FUNCTION_BLOCK FB_UpperFeedInConveyor EXTENDS FB_ObjectBase_V2
VAR_INPUT
	
	_fbDiameterMovement : REFERENCE TO FB_DiameterMovement;
	
	Cylinder 	: REFERENCE TO UNI_CylinderList;
	Motor	 	: REFERENCE TO UNI_MotorList;
	Input 	 	: REFERENCE TO ST_InputTable;
	OutPut	 	: REFERENCE TO ST_OutputTable;
	
	Info		: ST_Auto_UpperFeedInConveyorInfo;
	
	AddingBox	: BOOL;
//    Execute    :BOOL;   // True : This prog will start.
//    Abort      :BOOL;   // True : This prog will be abort.
//    Reset      :BOOL;   // True : This prog will be reset.
//    ObjectName :STRING; // Set this fb name(About it's action)
END_VAR

VAR_OUTPUT
//	Status		: ST_StatusBasic;
	FeedBack    : ST_Auto_UpperFeedInConveyorFeedback;	
	_bForceUpperCV_Use	: BOOL;	
//    Busy    :BOOL;        // True : This prog is running.
//    Done    :BOOL;        // True : Command has been executed.
//    Aborted :BOOL;        // True : This prog is aborted.
//    Error   :BOOL;        // True : This prog has an error.
//    ErrorID :UINT;       // Output ErrorID
//    Status  :T_MaxString; // Output this prog status by string(255bytes)
END_VAR

VAR
//    eState :E_MethodStatus_Basic;
//	uiExecutingStep : UDINT; // This var is used to been controll STATE_EXECUTING process.
//	uiResettingStep : UDINT;
//	uiAbortingStep : UDINT;
//	_Executed :BOOL; // Executing process completed.
//	_Error : BOOL; // FB has an error.
//	_ResetCompleted : BOOL; // FB resetting completed.
//	_AbortCompleted : BOOL; // FB aborting completed.
	_Abort		: BOOL;
	strStatus	: T_MaxString;
	uiResumeStep : UINT;
	iMoveConveyor	:INT;// 1 = MoveForward , -1 = Move reverse , 0 or other = Stop
	tonUpperConveyorTimeOut			:TON;
	tonUpperConveyorDelay			:TON;
	tonUpperTimeOut					:TON;
	tonUpperTimeOutFive 			:TON;
	tonWaitSecondBoxArriveTimeout 	:TON;
	tonFeedAirBlowtime 				:TON;
	tonReverseConveyorDelay			:TON;
	TON_CheckHaveBox				:TON ;
	NoFirstBoxDiameter : BOOL;
	SecondBox	:BOOL;
	bSecondBoxInCameraPos :BOOL;
	uiFirstBoxDiameterStep :UINT :=0;
	uiSecondBoxAirBlowStep :UINT :=0;
	_UniqueErrorCode :STRING;
	
	
	//record time for C# photo
	tRecordTimer 		: ARRAY [1..100] OF TIME;
	tRecordFirstTimer	: ARRAY [1..100] OF TIME;
	tRecordSecondTimer	: ARRAY [1..100] OF TIME;
	TON_RecordTimer 	: TON;
	TON_RecordFirstTimer		: TON ;
	TON_RecordSecondTimer		: TON;
	TSaveTime					: TIME;
	TSaveFirstTime				: TIME;
	TSaveSecondTime				: TIME;
	iArrayNumber 				: INT :=1;
	iResetNumber				: INT;
	bResetRecordInfo			: BOOL;
	
	
END_VAR

A00_BasicUnits();
SUPER^.A10_StateControl();

ACTION A00_BasicUnits:
tonUpperConveyorTimeOut(PT:=T#20S);
tonUpperConveyorDelay();
tonUpperTimeOut(PT:=T#5.0S);
tonUpperTimeOutfive(PT:=T#60S);
tonWaitSecondBoxArriveTimeout(PT:=T#20S);
tonFeedAirBlowtime(PT:=info.FeedAirblowTime);
tonReverseConveyorDelay(PT:=T#6S);
TON_CheckHaveBox(PT :=T#35S);
ErrorID :=2710;



TON_RecordTimer (PT:=T#1D);
TON_RecordFirstTimer (PT := T#1D);
TON_RecordSecondTimer (PT := T#1D);

// only for record the photo time use
IF bResetRecordInfo THEN
	FOR iResetNumber :=1 TO 100 DO
		tRecordTimer[iResetNumber] :=T#0S;
		tRecordFirstTimer[iResetNumber] :=T#0S;
		tRecordSecondTimer[iResetNumber] :=T#0S;
	END_FOR
END_IF
END_ACTION

METHOD GetModelState
VAR_OUTPUT
    xDone    :BOOL;
    xBusy    :BOOL;
    xError   :BOOL;
    xAborted :BOOL;
    iErrorID :UDINT;
	UniqueErrorCode : STRING;
END_VAR
xDone    := Done;
xBusy    := Busy;
xError   := Error;
xAborted := Abort;
iErrorID := ErrorID;
END_METHOD

METHOD GetName : STRING
GetName := ObjectName;
END_METHOD

METHOD  M_STATE_ABORTED
VAR_INPUT
END_VAR
ERROR :=TRUE;
Busy := FALSE;
Aborted := TRUE;
_Abort := FALSE;
UniqueErrorCode:=_UniqueErrorCode;
SUPER^.Status := strStatus;

IF NOT Execute THEN
	eSTATE:=STATE_RESETTING;
	
ELSIF Execute AND Reset THEN

		CASE uiExecutingStep OF
			20:
				uiExecutingStep :=10;
				strStatus :='prepare cylinders retry';
				
			100:
				uiExecutingStep :=100;
				strStatus :='check no box retry';
			200:
				uiExecutingStep :=200;
				strStatus :='check Block3Cylinder retry';

			400://將讀碼壓盒1 往後 重做一次
				Cylinder.List.fbUpCV_CamaraPress1.M_Retract();
				IF Cylinder.List.fbUpCV_CamaraPress1.InRearPosition THEN
				uiExecutingStep :=300;
				strStatus :='check ReadCodeBox1 infrontposition retry';
				END_IF
			460:	//Box1 done step abort
				uiExecutingStep :=450;
				strStatus :='Check FirstBoxCamaraDone info retry';
			550:
				uiExecutingStep :=500;
				strStatus :='ReadCodePressBox1Cylinder and FeedInBlockBox3Cylinder Backward retry';
			600:
				uiExecutingStep :=600;
				strStatus :='FirstBoxCameraDiameterRequest Info retry';
			610:
				uiExecutingStep :=610;
				strStatus :='CodeReadingBoxDetection first box leave retry';
			700:
				uiExecutingStep :=700;
				strStatus :='UpperFeedInBlockBox2Cylinder MoveForward retry';
			800:
				uiExecutingStep :=800;
				strStatus :='Box not at UpperBox2Detection retry ';
				
			1000:
				Cylinder.List.fbUpCV_DiameterPress.M_Retract();
				IF Cylinder.List.fbUpCV_DiameterPress.InRearPosition THEN
					uiExecutingStep :=800;
					strStatus :='DiameterMeasurementPressBoxCylinder MoveBackward retry';
				END_IF
			1200:
				Cylinder.List.fbUpCV_CamaraPress1.M_Retract();
				Cylinder.List.fbUpCV_CamaraPress2.M_Retract();
				IF Cylinder.List.fbUpCV_CamaraPress1.InRearPosition AND 
					Cylinder.List.fbUpCV_CamaraPress2.InRearPosition THEN
					uiExecutingStep :=1100;
					strStatus :='ReadCodePressBox 1 and 2 Cylinder retry';
				END_IF
			1300:
				uiExecutingStep :=1300;
				strStatus :='SecondBoxCameraDone info retry';
			1400:
				uiExecutingStep :=1400;
				strStatus :='FirstBoxCameraDiameterDone info retry';
			1600:
				uiExecutingStep :=1500;
				strStatus :='DiameterMeasurementPressBoxCylinder and FeedInBlockBox2Cylinder MoveBackward retry';
			1700:
				uiExecutingStep :=1700;
				strStatus :='check UpperBox2Detection have box';
			1800:
				Cylinder.List.fbUpCV_DiameterPress.M_Retract();
				IF Cylinder.List.fbUpCV_DiameterPress.InRearPosition THEN
				uiExecutingStep :=1700;
				strStatus :='DiameterMeasurementPressBoxCylinder Forward retry';
				END_IF
			1900:
				uiExecutingStep :=1900;
				strStatus :='DiameterMovement PickDone  retry';
			2000:
				uiExecutingStep :=2000;
				strStatus :='SecondBoxCameraDiameterDone retry';
			2100:	
				uiExecutingStep :=2100;
				strStatus :='_fbDiameterMovement done retry';
			2200:
				
				
		END_CASE
	
	eSTATE:=STATE_EXECUTING;
	
END_IF
END_METHOD

METHOD  M_STATE_ABORTING
VAR_INPUT
END_VAR
Busy :=FALSE;
CASE uiAbortingStep OF
	0:
		tonUpperConveyorTimeOut.IN 	:=FALSE;
		tonUpperConveyorDelay.IN	:=FALSE;
		tonUpperTimeOut.IN 			:=FALSE;
		tonUpperTimeOutfive.IN		:=FALSE;
		TON_CheckHaveBox.IN 		:=FALSE;
		uiAbortingStep :=100;
	100:
		Motor.List.UpCV.M_MotorStop();
		OutPut.bCamara_Blow :=FALSE;
		IF Motor.List.UpCV.InStopped THEN
			uiAbortingStep :=9999;
		END_IF
	9999:	
		_AbortCompleted:=TRUE;
END_CASE

IF _AbortCompleted THEN	
	eSTATE :=STATE_ABORTED;
END_IF
END_METHOD

METHOD  M_STATE_DONE
VAR_INPUT
END_VAR
Busy := FALSE;
Done:=TRUE;
_fbDiameterMovement.Execute := FALSE;
_fbDiameterMovement.bContinue:=FALSE;
IF NOT Execute THEN
	eSTATE:=STATE_RESETTING;
END_IF
END_METHOD

METHOD  M_STATE_DORMANT
VAR_INPUT
END_VAR
Busy    := FALSE;
Done    := FALSE;
Aborted := FALSE;
Error   := FALSE;
FeedBack.InterventionRequest :=FALSE;
strStatus :='No Error';
uiExecutingStep :=0;
uiResettingStep	:=0;
NoFirstBoxDiameter:= SecondBox:=FALSE;
tonUpperConveyorTimeOut.IN := FALSE;
tonUpperConveyorDelay.IN :=FALSE;
tonUpperTimeOut.IN :=FALSE;
tonUpperTimeOutFive.IN :=FALSE;
tonWaitSecondBoxArriveTimeout.IN :=FALSE;
TON_CheckHaveBox.IN :=false;
tonFeedAirBlowtime.IN :=false;
bSecondBoxInCameraPos := FALSE;
_bForceUpperCV_Use := false;
_Abort := _Executed := _Error:= _ResetCompleted:=_AbortCompleted:=FALSE;
iMoveConveyor := 0;
uiFirstBoxDiameterStep  :=0;
uiSecondBoxAirBlowStep	:=0;
_UniqueErrorCode :='0';
IF Execute THEN
	eSTATE:=STATE_EXECUTING;
END_IF
END_METHOD

METHOD  M_STATE_ERROR
VAR_INPUT
END_VAR
ERROR :=TRUE;
Busy :=FALSE;
UniqueErrorCode:=_UniqueErrorCode;
SUPER^.Status := strStatus;
_fbDiameterMovement.Execute := FALSE;


Motor.List.UpCV.M_MotorStop(); 
OutPut.bCamara_Blow :=FALSE;

IF NOT Execute THEN	
eSTATE:=STATE_RESETTING;
END_IF
END_METHOD

METHOD  M_STATE_EXECUTING
VAR_INPUT
END_VAR

VAR_INST
	
	
END_VAR
VAR
	END_I: INT;
	
END_VAR
Busy :=TRUE;

//Conveyor motor control
CASE iMoveConveyor OF
	1:
	Motor.list.UpCV.M_MoveForward();
	Cylinder.List.fbUpCV_CamaraPress4.M_Retract(); //Feedin working , open the end to allow box feedin
	//OutPut.bCamara_Blow :=TRUE;
	-1:
	Motor.list.UpCV.M_MoveBackward();
	Cylinder.List.fbUpCV_CamaraPress4.M_Retract(); //Feedin working , open the end to allow box feedin
ELSE		
	Motor.list.UpCV.M_MotorStop();
	Cylinder.List.fbUpCV_CamaraPress4.M_Extend();// End feedin , block the conveyor in case no one push boxes in working area
	//OutPut.bCamara_Blow :=FALSE;		change use airflow to take photo before
END_CASE



CASE uiExecutingStep OF
	
0 : // StandBy
	TON_RecordTimer.IN := TRUE;
	iMoveConveyor:=0;
	tonUpperConveyorTimeOut.IN:=FALSE;
	tonUpperConveyorDelay.IN :=FALSE;
	tonUpperConveyorDelay.PT:=T#200MS;
	IF Info.NrOfBox=1 THEN
		SecondBox:=FALSE;
	ELSIF Info.NrOfBox=2 THEN
		SecondBox:=TRUE;	
	ELSE
	_Error := TRUE;
	  strStatus := 'Data not correct';		
	END_IF
	uiExecutingStep :=10;

10: //Prepare cylinders
	IF Cylinder.List.fbUpCV_FeedInPress1.xError THEN
		Cylinder.List.fbUpCV_FeedInPress1.M_Reset();
	END_IF
	IF Cylinder.List.fbUpCV_FeedInPress2.xError THEN
		Cylinder.List.fbUpCV_FeedInPress1.M_Reset();
	END_IF
	IF Cylinder.List.fbUpCV_DiameterPress.xError THEN
		Cylinder.List.fbUpCV_DiameterPress.M_Reset();
	END_IF
	IF Cylinder.List.fbUpCV_CamaraPress1.xError THEN
		Cylinder.List.fbUpCV_CamaraPress1.M_Reset();
	END_IF
	IF Cylinder.List.fbUpCV_CamaraPress2.xError THEN
		Cylinder.List.fbUpCV_CamaraPress2.M_Reset();
	END_IF
	IF Cylinder.List.fbUpCV_CamaraPress4.xError THEN
		Cylinder.List.fbUpCV_CamaraPress4.M_Reset();
	END_IF
	IF Cylinder.List.fbUpCV_Block1.xError THEN
		Cylinder.List.fbUpCV_Block1.M_Reset();
	END_IF
	IF Cylinder.List.fbUpCV_Block2.xError THEN
		Cylinder.List.fbUpCV_Block2.M_Reset();
	END_IF
	IF Cylinder.List.fbUpCV_Block3.xError THEN
		Cylinder.List.fbUpCV_Block3.M_Reset();
	END_IF
	IF Motor.List.UpCV.xError THEN
		Motor.List.UpCV.M_Reset();
	END_IF
	
	uiExecutingStep :=20;
	
20: //Prepare cylinders
	tonUpperTimeOut.IN :=TRUE;
	Cylinder.List.fbUpCV_FeedInPress1.M_Retract();		(* Cylinder.List.fbUpCV_FeedInPress1.M_Retract();*)	
	Cylinder.List.fbUpCV_FeedInPress2.M_Retract();		(*Cylinder.List.fbUpCV_FeedInPress2.M_Retract();*)
	Cylinder.List.fbUpCV_DiameterPress.M_Retract();		(*Cylinder.List.fbUpCV_DiameterPress.M_Retract();*)
	Cylinder.List.fbUpCV_CamaraPress1.M_Retract();		(*Cylinder.List.fbUpCV_CamaraPress1.M_Retract();*)		
	//Cylinder.List.fbUpCV_CamaraPress2.M_Retract();	(*Cylinder.List.fbUpCV_CamaraPress2.M_Retract();*)
	Cylinder.List.fbUpCV_CamaraPress4.M_Retract();		(*Cylinder.List.fbUpCV_CamaraPress4.M_Retract();*)	
	Cylinder.List.fbUpCV_Block1.M_Retract();			(*Cylinder.List.fbUpCV_Block1.M_Retract();*)
	Cylinder.List.fbUpCV_Block2.M_Retract();			(*Cylinder.List.fbUpCV_Block2.M_Retract();*)
	Cylinder.List.fbUpCV_Block3.M_Retract();			(*Cylinder.List.fbUpCV_Block3.M_Retract();*)

	//edit by Min 20250326
	IF Cylinder.List.fbUpCV_FeedInPress1.InRearPosition AND		
		Cylinder.List.fbUpCV_FeedInPress2.InRearPosition AND
		Cylinder.List.fbUpCV_DiameterPress.InRearPosition AND
		Cylinder.List.fbUpCV_CamaraPress1.InRearPosition AND
		Cylinder.List.fbUpCV_CamaraPress4.InRearPosition AND
		Cylinder.List.fbUpCV_Block1.InRearPosition AND
		Cylinder.List.fbUpCV_Block2.InRearPosition AND
		Cylinder.List.fbUpCV_Block3.InRearPosition THEN
		
		tonUpperTimeOut.IN :=FALSE;
		uiExecutingStep :=100;	
	END_IF
	IF tonUpperTimeOut.Q THEN
		_Abort :=TRUE;
		strStatus :='Prepare Cylinder clear command timeout';
	END_IF
	
100:// Check No Box 
	IF Input.bUpCV_Block1Detect_Sensor OR 
	  Input.bUpCV_Block2Detect_Sensor OR
	  Input.bUpCV_BoxArrived_Sensor OR
	  Input.bUpCV_Block3Detect_Sensor THEN
	 	 IF NOT AddingBox THEN
		 _bForceUpperCV_Use := TRUE;		//force UpperCV for Backward CV use
	 	 uiExecutingStep :=110; //Try reverse conveyor 
			ELSE 
			  _Abort := TRUE;
		 	 strStatus := 'Conveyor not ready , please remove boxes in front';
		  END_IF
	 ELSE
 		uiExecutingStep :=200; 
	 END_IF
110:
		iMoveConveyor:= -1;
		Cylinder.List.fbUpCV_CamaraPress2.M_Retract();
		tonReverseConveyorDelay.IN :=TRUE;
		uiExecutingStep :=120;

120:
		//tonFeedAirBlowtime.IN :=TRUE;
		IF tonReverseConveyorDelay.Q THEN
			iMoveConveyor :=0;
			uiExecutingStep :=130; 
		END_IF
130:
		tonReverseConveyorDelay.IN :=FALSE;
		IF Input.bUpCV_Block1Detect_Sensor OR 
		  Input.bUpCV_Block2Detect_Sensor OR
		  Input.bUpCV_BoxArrived_Sensor OR
	 	 Input.bUpCV_Block3Detect_Sensor THEN 
			  _Abort := TRUE;
		 	 strStatus := 'Conveyor not ready , please remove boxes in front';
		 ELSE
			uiExecutingStep :=140; 	 
		 END_IF		
140:
   		IF Motor.list.UpCV.InStopped THEN
			uiExecutingStep :=200;
		END_IF
200: // motor start and camera block up 
	_bForceUpperCV_Use := FALSE;		//release UpperCV force use 
	tonUpperConveyorTimeOut.IN:=TRUE;
	iMoveConveyor:=1;
	Cylinder.List.fbUpCV_CamaraPress2.M_Retract();
	Cylinder.List.fbUpCV_Block3.M_Extend();
	IF Cylinder.List.fbUpCV_Block3.InFrontPosition AND
		Cylinder.List.fbUpCV_CamaraPress2.InRearPosition THEN
		tonUpperConveyorTimeOut.IN:=FALSE;
		uiExecutingStep :=300;
	END_IF
	IF tonUpperConveyorTimeOut.Q THEN
	  _Error := TRUE;
	  strStatus := 'Cylinder.List.fbUpCV_Block3 timeout';
	END_IF
		  
	  
300://Dtect camera sensor and wait first box arrive in camera position
	TON_CheckHaveBox.IN :=TRUE;
	tonUpperConveyorDelay.IN:=Input.bUpCV_Block3Detect_Sensor; //Delay a moment to make sure box move till end of block 	
	IF tonUpperConveyorDelay.Q THEN
			TON_CheckHaveBox.IN :=FALSE;
			Cylinder.List.fbUpCV_CamaraPress1.M_Extend(); //Press box 
			tonUpperConveyorDelay.IN := FALSE;
			uiExecutingStep :=400;			
	END_IF
	IF TON_CheckHaveBox.Q THEN	//if behind not have box feedback box = 0
		uiExecutingStep := 2700;
	END_IF
	
400:// Check pressing job done for first box in camera position	
	tonUpperTimeOut.IN :=TRUE;
	IF Cylinder.List.fbUpCV_CamaraPress1.InFrontPosition THEN
		tonUpperTimeOut.IN := FALSE;
		Cylinder.List.fbUpCV_CamaraPress2.M_Extend();
		uiExecutingStep :=450;		
	END_IF
	IF tonUpperTimeOut.Q THEN
		_Abort := TRUE;
		strStatus := 'Cylinder.List.fbUpCV_CamaraPress1.M_MoveForward timeout';
	END_IF

450:// send first box camera signal
	
	tonFeedAirBlowtime.IN :=TRUE;
	OutPut.bCamara_Blow :=TRUE;
	IF tonFeedAirBlowtime.Q THEN
		tonFeedAirBlowtime.IN:=FALSE;
		OutPut.bCamara_Blow :=FALSE;
		FeedBack.FirstBoxCamera :=TRUE;
		TON_RecordFirstTimer.IN :=TRUE;
		uiExecutingStep :=460;
	END_IF
	

460: // Wait first box camera done
	// todo : timeout
	tonUpperTimeOutFive.IN :=TRUE;		//T#5S
	IF Info.FirstBoxCameraDone THEN
		tonUpperTimeOutFive.IN :=FALSE;
		FeedBack.FirstBoxCamera :=FALSE;
		uiExecutingStep :=500;
	END_IF	
	IF tonUpperTimeOutFive.Q THEN
		_Abort :=TRUE;
		strStatus := 'C# FirstBoxCameraDone timeout';
	END_IF
	
500://Let first box move forward
	TSaveFirstTime 	:= TON_RecordFirstTimer.ET;
	TON_RecordFirstTimer .IN :=FALSE;
	Cylinder.List.fbUpCV_CamaraPress1.M_Retract(); // release press
	Cylinder.List.fbUpCV_Block3.M_Retract();//release blocker todo : add description
	uiExecutingStep :=550;
	
550://check cylinder inrearposition		edit by Min 20250326
	tonUpperTimeOut.IN :=TRUE;
	IF Cylinder.List.fbUpCV_CamaraPress1.InRearPosition AND		
		Cylinder.List.fbUpCV_Block3.InRearPosition THEN
		
		uiExecutingStep :=600;
	END_IF
	IF tonUpperTimeOut.Q THEN
		_Abort := TRUE;
		strStatus := 'Cylinder.List.fbUpCV_CamaraPress1 or Cylinder.List.fbUpCV_Block3 InRearPosition timeout';
	END_IF
	
600://Check if diameter camera needed
	tonUpperTimeOut.IN :=FALSE;
	tonUpperTimeOutFive.IN :=TRUE;
	IF Info.FirstBoxCameraDiameterRequest THEN
		tonUpperTimeOutFive.IN :=FALSE;
		uiExecutingStep :=700;
		ELSE
			IF SecondBox THEN
				tonUpperTimeOutFive.IN :=FALSE;
				NoFirstBoxDiameter:=TRUE;
				uiExecutingStep :=610;//Only if box 1 no need to measure diameter
			ELSE
				tonUpperTimeOutFive.IN :=FALSE;
				uiExecutingStep :=2400;	
			END_IF
	END_IF
	IF tonUpperTimeOutFive.Q THEN
		_Abort := TRUE;
		strStatus :='C# FirstBoxCameraDiameterRequest timeout';
	END_IF
	
610: //Check Box 1 leave read code camera position
	tonUpperTimeOut.IN :=TRUE;
	tonUpperConveyorDelay.IN := NOT Input.bUpCV_Block3Detect_Sensor;
	IF tonUpperConveyorDelay.Q THEN
		tonUpperConveyorDelay.IN :=FALSE;
		uiExecutingStep :=620;
	END_IF
	IF tonUpperTimeOut.Q  THEN
		_Abort :=TRUE;
		strStatus :='Input.bUpCV_Block3Detect_Sensor first box leave timeout';
	END_IF
	
620: // Leave Box 2				//timeout and Check InRearPositonEdit by Min 20250326	
		tonUpperTimeOut.IN :=FALSE;	
		IF SecondBox THEN			
			Cylinder.List.fbUpCV_CamaraPress2.M_Retract(); //Release press box
			Cylinder.List.fbUpCV_Block3.M_Extend(); //release blocker
			IF Cylinder.List.fbUpCV_CamaraPress2.InRearPosition AND Cylinder.List.fbUpCV_Block3.InFrontPosition THEN
				uiExecutingStep :=1100;
			END_IF
		END_IF
		
700: //Rise diameter blocker
	tonUpperTimeOut.IN :=TRUE;
	Cylinder.List.fbUpCV_Block2.M_Extend();
	IF Cylinder.List.fbUpCV_Block2.InFrontPosition THEN
		tonUpperTimeOut.IN :=FALSE;
		uiExecutingStep :=800;
	END_IF
	IF tonUpperTimeOut.Q THEN
		_Abort :=TRUE;
		strStatus :='Cylinder.List.fbUpCV_Block2 MoveForward timeout';
	END_IF
800: // wait first box ready on diameter position
	tonUpperTimeOut.IN :=TRUE;
	tonUpperConveyorDelay.IN:=Input.bUpCV_Block2Detect_Sensor;
	IF tonUpperConveyorDelay.Q THEN
		tonUpperTimeOut.IN :=FALSE;
		tonUpperConveyorDelay.IN:=FALSE;
		Cylinder.List.fbUpCV_DiameterPress.M_Extend();
		
		IF SecondBox THEN	
			tonUpperTimeOut.IN :=FALSE;		
			Cylinder.List.fbUpCV_CamaraPress2.M_Retract();
			Cylinder.List.fbUpCV_Block3.M_Extend();
		END_IF
		uiExecutingStep :=1000;
	END_IF
	IF tonUpperTimeOut.Q THEN
		_Abort :=TRUE;
		strStatus :='Box not at Input.bUpCV_Block2Detect_Sensor ';
	END_IF
	
1000: // Wait diameter blocker ready
	tonUpperTimeOut.IN :=TRUE;
	IF 	Cylinder.List.fbUpCV_DiameterPress.InFrontPosition THEN
		tonUpperTimeOut.IN :=FALSE;
		uiExecutingStep :=1100;
	END_IF
	IF tonUpperTimeOut.Q THEN
		_Abort :=TRUE;
		strStatus :='Cylinder.List.fbUpCV_DiameterPress MoveForward timeout';
	END_IF

1100: // Pick needle to diameter camera

		
		CASE uiFirstBoxDiameterStep OF
			
		0:
			IF NOT NoFirstBoxDiameter THEN
	  			_fbDiameterMovement.Execute := TRUE;
				uiFirstBoxDiameterStep:=100;
			ELSE
				uiFirstBoxDiameterStep:=9000;	
	  		END_IF
		
		100:
			IF _fbDiameterMovement.Busy THEN
				uiFirstBoxDiameterStep:=200;
			END_IF	
			
		200:
			tonUpperTimeOutFive.IN :=TRUE;
			 IF _fbDiameterMovement.PickDone THEN
				  tonUpperTimeOutFive.IN :=FALSE;
				  FeedBack.FirstBoxCameraDiameter:=TRUE;		  
			  END_IF
			 IF Info.FirstBoxCameraDiameterDone THEN
				tonUpperTimeOutFive.IN:=FALSE;
				 FeedBack.FirstBoxCameraDiameter:=FALSE;
			 	_fbDiameterMovement.bContinue:=TRUE;
			 	uiFirstBoxDiameterStep:=300;
			  END_IF
			 IF tonUpperTimeOutFive.Q THEN
				 _Error :=TRUE;
				 strStatus :='box1 diameter timeout';
			 END_IF
		300:
			 IF _fbDiameterMovement.Done THEN
				  uiFirstBoxDiameterStep:=9000;		  
			  END_IF	  
		
		9000:
				_fbDiameterMovement.bContinue:=FALSE;
				_fbDiameterMovement.Execute:=FALSE;
				Cylinder.List.fbUpCV_DiameterPress.M_Retract();
				Cylinder.List.fbUpCV_Block2.M_Retract();
				// first box leave	  
				
				IF bSecondBoxInCameraPos AND 
					Cylinder.List.fbUpCV_DiameterPress.InRearPosition AND
					Cylinder.List.fbUpCV_Block2.InRearPosition THEN
					
					uiExecutingStep :=1200;
				END_IF
		END_CASE
						
		
	  		IF SecondBox THEN
				tonWaitSecondBoxArriveTimeout.IN :=TRUE;
	  			tonUpperConveyorDelay.IN := Input.bUpCV_Block3Detect_Sensor;
 				IF tonUpperConveyorDelay.Q THEN								
					tonUpperConveyorDelay.IN:=FALSE;
					tonWaitSecondBoxArriveTimeout.IN :=FALSE;
					Cylinder.List.fbUpCV_CamaraPress2.M_Extend();
					Cylinder.List.fbUpCV_CamaraPress1.M_Extend();
//					bSecondBoxInCameraPos :=TRUE;
				END_IF	
	 		 ELSE
				 bSecondBoxInCameraPos:=TRUE;
	 		 END_IF
			 
		CASE uiSecondBoxAirBlowStep OF
			 0:
			 	IF 	Cylinder.List.fbUpCV_CamaraPress1.InFrontPosition AND 
					Cylinder.List.fbUpCV_CamaraPress2.InFrontPosition THEN
						uiSecondBoxAirBlowStep :=10;
				END_IF
			10:
				OutPut.bCamara_Blow :=TRUE;		//take photo need airflow before
				tonFeedAirBlowtime.IN :=TRUE;
					IF tonFeedAirBlowtime.Q THEN		
						tonFeedAirBlowtime.IN :=FALSE;
						OutPut.bCamara_Blow :=FALSE;
						FeedBack.SecondBoxCamera:=TRUE;
						TON_RecordSecondTimer.IN :=TRUE;
						uiSecondBoxAirBlowStep :=20;
					END_IF
			20:
				IF Info.SecondBoxCameraDone THEN
					uiSecondBoxAirBlowStep :=30;
					TSaveSecondTime := TON_RecordSecondTimer.ET;
				END_IF
			30:	
					
					
					TON_RecordSecondTimer.IN :=FALSE;
					bSecondBoxInCameraPos:=TRUE;	
			
		END_CASE
		
//			IF Cylinder.List.fbUpCV_CamaraPress1.InFrontPosition AND 
//				Cylinder.List.fbUpCV_CamaraPress2.InFrontPosition THEN
//				OutPut.bCamara_Blow :=TRUE;		//take photo need airflow before
//				tonFeedAirBlowtime.IN :=TRUE;
//					IF tonFeedAirBlowtime.Q THEN		
//						tonFeedAirBlowtime.IN :=FALSE;
//						OutPut.bCamara_Blow :=FALSE;
//						FeedBack.SecondBoxCamera:=TRUE;	
//							IF Info.SecondBoxCameraDone THEN
//								bSecondBoxInCameraPos:=TRUE;	
//							END_IF	
//					END_IF
//			END_IF
	  
	  IF tonUpperConveyorTimeOut.Q THEN
			_Error :=TRUE;
			strStatus:='First box diameter timeout';		
		  
	  END_IF
		IF tonWaitSecondBoxArriveTimeout.Q THEN
			IF Input.bUpCV_ReLoadDetect_Sensor THEN
				_Error :=TRUE;
				strStatus:='Second box feedin to read code camera pos timeout';		
			ELSE
				tonUpperConveyorTimeOut.IN :=FALSE;
				SecondBox :=FALSE;
			END_IF	 
		END_IF

1200: 	// If first box leave diameter sensor , let second box go
		tonUpperTimeOut.IN :=TRUE;
		tonUpperConveyorDelay.PT:=T#600MS;		
		tonUpperConveyorDelay.IN := NOT Input.bUpCV_Block2Detect_Sensor;
		
		IF tonUpperConveyorDelay.Q THEN
			tonUpperConveyorDelay.IN :=FALSE;
			tonUpperTimeOut.IN :=FALSE;
			IF SecondBox AND INfo.SecondBoxCameraDiameterRequest THEN
				tonUpperTimeOut.IN :=FALSE;
				Cylinder.List.fbUpCV_Block2.M_Extend();
				Cylinder.List.fbUpCV_CamaraPress1.M_Retract();
				Cylinder.List.fbUpCV_Block3.M_Retract();
				uiExecutingStep :=1700;
			ELSE
				tonUpperTimeOut.IN :=FALSE;
				uiExecutingStep :=2400;	
			END_IF

		END_IF
		IF tonUpperTimeOut.Q THEN
			_Abort :=TRUE;
			strStatus :='First box still at Input.bUpCV_Block2Detect_Sensor';
		END_IF

1700: //Second box diameter request
		tonUpperTimeOut.IN :=TRUE;
		tonUpperConveyorDelay.IN :=Input.bUpCV_Block2Detect_Sensor;
		IF tonUpperConveyorDelay.Q THEN
			tonUpperTimeOut.IN :=FALSE;
			tonUpperConveyorDelay.IN :=FALSE;
			Cylinder.List.fbUpCV_DiameterPress.M_Extend();
			uiExecutingStep :=1800;
		END_IF
		IF tonUpperTimeOut.Q THEN
			_Abort :=TRUE;
			strStatus :='Input.bUpCV_Block2Detect_Sensor not have box';
		END_IF
1800: //wait second box in diameter position
		tonUpperTimeOut.IN :=TRUE;
		IF Cylinder.List.fbUpCV_DiameterPress.InFrontPosition THEN
			tonUpperTimeOut.IN :=FALSE;
			uiExecutingStep :=1900;
		END_IF
		IF tonUpperTimeOut.Q THEN
			_Abort :=TRUE;
			strStatus :='Cylinder.List.fbUpCV_DiameterPress MoveForward timeout';
			
		END_IF
		
1900:
		tonUpperTimeOutFive.IN :=TRUE;
		_fbDiameterMovement.Execute :=TRUE	;	
		IF _fbDiameterMovement.PickDone THEN
			tonUpperTimeOutFive.IN :=FALSE;
			FeedBack.SecondBoxCameraDiameter:=TRUE;
			uiExecutingStep :=2000;
		END_IF
		IF tonUpperTimeOutFive.Q THEN
			_Abort :=TRUE;
			strStatus :='C# DiameterMovement Pickdone timeout';
		END_IF
2000:	//check Second Box CamaraDone
		tonUpperTimeOutFive.IN :=TRUE;
		IF info.SecondBoxCameraDiameterDone THEN
			tonUpperTimeOutFive.IN :=FALSE;
			FeedBack.SecondBoxCameraDiameter:=FALSE;
			_fbDiameterMovement.bContinue:=TRUE;
			uiExecutingStep :=2100;
		END_IF
		IF tonUpperTimeOutFive.Q THEN
			_Abort :=TRUE;
			strStatus :='C# SecondBoxCameraDiameterDone timeout';
		END_IF		
2100:	
		tonUpperTimeOutFive.IN :=TRUE;
		IF _fbDiameterMovement.Done THEN
			tonUpperTimeOutFive.IN :=FALSE;
			_fbDiameterMovement.Execute:=FALSE;
			uiExecutingStep :=2150;
		END_IF
		IF tonUpperTimeOutFive.Q THEN
			_Abort :=TRUE;
			strStatus :='_fbDiameterMovement Done timeout';
		END_IF
2150:
		IF  Input.bUpCV_BoxArrived_Sensor  AND 
			NOT Input.bUpCV_Block1Detect_Sensor  THEN
			uiExecutingStep :=2200;
		END_IF
2200:	// release box 2 from diameter camera pos
		tonUpperTimeOut.IN :=TRUE;
		tonUpperConveyorDelay.PT:=T#100MS;
		tonUpperConveyorDelay.IN := NOT Input.bUpCV_Block1Detect_Sensor ;
		IF tonUpperConveyorDelay.Q THEN	
			tonUpperConveyorDelay.IN := FALSE;
			Cylinder.List.fbUpCV_Block1.M_Extend();
			Cylinder.List.fbUpCV_DiameterPress.M_Retract();		
			Cylinder.List.fbUpCV_Block2.M_Retract();
			uiExecutingStep :=2300;
		END_IF
		IF tonUpperTimeOut.Q THEN
			_Error :=TRUE;
			strStatus := 'There is a box on Input.bUpCV_Block1Detect_Sensor '; 
		END_IF
		
		
2300:
		tonUpperTimeOut.IN :=TRUE;
		IF 	Cylinder.List.fbUpCV_DiameterPress.InRearPosition AND
			Cylinder.List.fbUpCV_Block1.InFrontPosition AND
			Cylinder.List.fbUpCV_Block2.InRearPosition THEN
			tonUpperTimeOut.IN :=FALSE;
			uiExecutingStep :=2500;
		END_IF	
		IF tonUpperTimeOut.Q THEN
			_Error :=TRUE;
			strStatus :='BlockBox1 MoveForward or BlockBox2 MoveBackward or DiameterMeasurementPressBox MoveBackward timeout';
		END_IF
2400:	//Check Box1 in FeedInBox1Detecting and Box2 leave BlockBox2Detecting
		
		tonUpperConveyorDelay.PT:=T#200MS;
		tonUpperConveyorDelay.IN := Input.bUpCV_BoxArrived_Sensor ;
		
		IF  tonUpperConveyorDelay.Q AND NOT Input.bUpCV_Block1Detect_Sensor  THEN
			tonUpperConveyorDelay.IN:=FALSE;
			Cylinder.List.fbUpCV_CamaraPress1.M_Retract();
			Cylinder.List.fbUpCV_Block3.M_Retract();
			Cylinder.List.fbUpCV_Block1.M_Extend();
			uiExecutingStep :=2500;
		END_IF
		
2500:	// Check Box1 in FeedInBox1Sensor and Box2 in BlockBox1Sensor
		tonUpperTimeOutFive.IN :=TRUE;
		tonUpperConveyorDelay.PT:=T#1000MS;
		tonUpperConveyorDelay.IN := Input.bUpCV_BoxArrived_Sensor  AND 
		(Input.bUpCV_Block1Detect_Sensor  OR NOT SecondBox);
		
		IF tonUpperConveyorDelay.Q THEN
			tonUpperTimeOutFive.IN :=FALSE;
			tonUpperConveyorDelay.IN :=FALSE;
			Cylinder.List.fbUpCV_FeedInPress1.M_Extend();
			IF SecondBox THEN
				Cylinder.List.fbUpCV_FeedInPress2.M_Extend();
			END_IF
			uiExecutingStep :=2600;
		END_IF
		IF tonUpperTimeOutFive.Q THEN
			_Error :=TRUE;
			strStatus :='FeedInBox1Detecting not have a box';
		END_IF
2600:
		tonUpperConveyorDelay.PT:=T#500MS;
		tonUpperTimeOut.IN := TRUE;
		tonUpperConveyorDelay.IN :=  Cylinder.List.fbUpCV_FeedInPress1.InFrontPosition AND
		 (Cylinder.List.fbUpCV_FeedInPress2.InFrontPosition OR NOT SecondBox);		
//		IF tonUpperConveyorDelay.IN THEN
//			iMoveConveyor:=0;
//			//Motor.list.UpCV.M_StopMotor();
//		END_IF
		IF tonUpperConveyorDelay.Q THEN
			iMoveConveyor:=0;
			tonUpperTimeOut.IN :=FALSE;
			tonUpperConveyorDelay.IN :=FALSE;
			 Cylinder.List.fbUpCV_FeedInPress1.M_Retract();
			IF SecondBox THEN
				Cylinder.List.fbUpCV_FeedInPress2.M_Retract();
			END_IF
			uiExecutingStep :=2700;
		END_IF	
		IF tonUpperTimeOut.Q THEN
			_Error :=TRUE;
			strStatus :=' Cylinder.List.fbUpCV_FeedInPress1 or Cylinder.List.fbUpCV_FeedInPress2 MoveForward timeout';
		END_IF
2700:
		tonUpperTimeOut.IN :=TRUE;
		IF TON_CheckHaveBox.IN THEN	// conveyor behind not have box feedback 0
			FeedBack.ActualNrOfBox:=0;
		ELSIF SecondBox THEN
			FeedBack.ActualNrOfBox:=2;
			ELSE
			FeedBack.ActualNrOfBox:=1;	
		END_IF
		//Cylinder.List.fbUpCV_Block1.M_Retract();
		//Cylinder.List.fbUpCV_CamaraPress2.M_Retract();
		IF NOT input.bUpCV_ReLoadDetect_Sensor  THEN
			FeedBack.InterventionRequest :=TRUE;
		END_IF
		IF// Cylinder.List.fbUpCV_Block1.InRearPosition AND
			 Cylinder.List.fbUpCV_FeedInPress1.InRearPosition AND
			Cylinder.List.fbUpCV_FeedInPress2.InRearPosition THEN
			//Cylinder.List.fbUpCV_CamaraPress2.InRearPosition THEN
			tonUpperTimeOut.IN :=FALSE;
			uiExecutingStep := 2800;
		END_IF	
		IF tonUpperTimeOut.Q THEN 
			_Error :=TRUE;
			strStatus :='FeedInPressBox1Cylinder or FeedInPressBox2Cylinder or ReadCodePressBox2Cylinder MoveBackward timeout';
		END_IF
		
2800:	//TO check the camera photo speed recoeding time
	TSaveTime 		:= TON_RecordTimer.ET;
	tRecordTimer[iArrayNumber] 			:=TSaveTime;
	tRecordFirstTimer[iArrayNumber] 	:=TSaveFirstTime;
	tRecordSecondTimer[iArrayNumber] 	:=TSaveSecondTime;
	uiExecutingStep := 2900;
2900:
	iArrayNumber := iArrayNumber+1;
	TON_RecordTimer.IN := FALSE;
	IF iArrayNumber >= 101 THEN
		bResetRecordInfo 	:=TRUE;
		iArrayNumber 		:=1;
	END_IF
	uiExecutingStep := 9999;
9999:
	bResetRecordInfo :=FALSE;
	TON_CheckHaveBox.IN :=FALSE;
	_Executed := TRUE;
				
END_CASE
	
	
IF NOT Execute THEN
	eState:=STATE_RESETTING;
END_IF
IF _Error THEN
	//FUN_UniqueErrorCodeGenerator(iErrorID := ErrorID,UinqueErrorCode=>_UniqueErrorCode);
	eState:=STATE_ERROR;
END_IF
IF _Abort OR Abort THEN
	//FUN_UniqueErrorCodeGenerator(iErrorID := ErrorID,UinqueErrorCode=>_UniqueErrorCode);
	eSTATE:=STATE_ABORTING;
END_IF
IF _Executed THEN
	eSTATE:=STATE_Done;
END_IF
END_METHOD

METHOD  M_STATE_RESETTING
VAR_INPUT
END_VAR
Error :=_Error;
Done :=_Executed;

tonUpperTimeOut.IN:=TRUE;
Motor.List.UpCV.M_MotorStop();

IF tonUpperTimeOut.Q OR NOT _Error THEN
	CASE uiResettingStep OF
		0: 
			IF _Error THEN
				Cylinder.List.fbUpCV_Block1.M_Retract();
			END_IF
			Cylinder.List.fbUpCV_FeedInPress1 .M_Retract();	
			Cylinder.List.fbUpCV_FeedInPress2.M_Retract();
			Cylinder.List.fbUpCV_DiameterPress.M_Retract();
			Cylinder.List.fbUpCV_CamaraPress1.M_Retract();	
			//UpperReadCodePressBox2Cylinder.M_Retract();	
			Cylinder.List.fbUpCV_Block2.M_Retract();	
			Cylinder.List.fbUpCV_Block3.M_Retract();	
			Cylinder.List.fbUpCV_CamaraPress4.M_Retract();
			OutPut.bCamara_Blow :=FALSE;
			_fbDiameterMovement.Execute := FALSE;
			_fbDiameterMovement.bContinue:=FALSE;
			FeedBack.InterventionRequest :=FALSE;
			FeedBack.FirstBoxCamera :=FALSE;
			FeedBack.FirstBoxCameraDiameter :=FALSE;
			FeedBack.SecondBoxCamera :=FALSE;
			FeedBack.SecondBoxCameraDiameter :=FALSE;

		
			uiResettingStep:=9999;
		
		9999:
			_ResetCompleted:=TRUE;
	END_CASE
END_IF
IF _ResetCompleted THEN
	eSTATE:=STATE_DORMANT;
END_IF
END_METHOD

END_FUNCTION_BLOCK

(* stored: Version 1.1.0.1, ProductVersion 3.1.4024.13
   POU FB_UpperFeedInConveyor: Id {b0a556d7-089b-4e5b-aece-2c8080fbc489}, SpecialFunc None
   Folder STATE: Id {336cf81a-2c47-4070-b1e8-3558b4c1b362}
   Action A00_BasicUnits: Id {163a9f76-8838-42a7-b540-e0044259cf51}
   Method GetModelState: Id {9b42938f-350f-451a-8071-11871af4efb1}
   Method GetName: Id {7be0ee6f-608b-4144-ab7b-2a2f1f70d1f5}
   Method M_STATE_ABORTED: Id {918c5246-ceda-4178-a0a7-4351a059cea2}
   Method M_STATE_ABORTING: Id {26e98244-888a-4eba-ab5f-389cbf7bce1d}
   Method M_STATE_DONE: Id {d1a4719c-7158-4715-ba72-a8c583af65bb}
   Method M_STATE_DORMANT: Id {3459b760-fe7c-4c55-8059-b4d0eae28804}
   Method M_STATE_ERROR: Id {00c69e48-07db-457b-8693-e90831a0e139}
   Method M_STATE_EXECUTING: Id {f86b848f-6f5f-4ca8-b816-5ea6b75940a7}
   Method M_STATE_RESETTING: Id {3adabedc-2b68-41f5-a609-d400b8b936b3} *)
